// ---- DUTs/IO/Topology/Term_1047_EK1100_7ACEE53D.TcDUT
{attribute 'GeneratedUsingTerminal: EK1100-0000-0018'}
{attribute addProperty BoxType "EK1100-0000-0018"}
{attribute addProperty Id "Term_1048_EL1809EL1809_32157CFD20Term_1049_EL1809EL1809_32157CFD20Term_1050_EL1809EL1809_32157CFD20Term_1051_EL1809EL1809_32157CFD20Term_1052_EL1809EL1809_32157CFD20Term_1053_EL1809EL1809_32157CFD20Term_1054_EL1809EL1809_32157CFD20Term_1055_EL1809EL1809_32157CFD20Term_1056_EL1809EL1809_32157CFD20Term_1057_EL1809EL1809_32157CFD20Term_1058_EL1809EL1809_32157CFD20Term_1059_EL1809EL1809_32157CFD20Term_1060_EL1809EL1809_32157CFD20Term_1061_EL1809EL1809_32157CFD20Term_1062_EL1809EL1809_32157CFD20Term_1063_EL1809EL1809_32157CFD20Term_1064_EL1809EL1809_32157CFD20Term_1065_EL1809EL1809_32157CFD20Term_1066_EL1809EL1809_32157CFD20Term_1068_EL1809EL1809_32157CFD20Term_1069_EL1809EL1809_32157CFD20Term_1070_EL1809EL1809_32157CFD20Term_1072_EL1809EL1809_32157CFD20Term_1073_EL1809EL1809_32157CFD20Term_1076_EL1809EL1809_32157CFD20Term_1077_EL1809EL1809_32157CFD20Term_1078_EL1809EL1809_32157CFD20Term_1081_EL1809EL1809_32157CFD20Term_1082_EL1809EL1809_32157CFD20Term_1083_EL1809EL1809_32157CFD20Term_1084_EL1809EL1809_32157CFD20Term_1085_EL1809EL1809_32157CFD20Term_1086_EL1809EL1809_32157CFD20Term_1087_EL1809EL1809_32157CFD20Term_1088_EL1809EL1809_32157CFD20Term_1089_EL1809EL1809_32157CFD20Term_1090_EL1809EL1809_32157CFD20Term_1091_EL1809EL1809_32157CFD20Term_1092_EL1809EL1809_32157CFD20Term_1093_EL1809EL1809_32157CFD20Term_1094_EL1809EL1809_32157CFD20Term_1095_EL1809EL1809_32157CFD20Term_1096_EL1809EL1809_32157CFD20Term_1097_EL1809EL1809_32157CFD20Term_1098_EL1809EL1809_32157CFD20Term_1099_EL1809EL1809_32157CFD20Term_1100_EL1809EL1809_32157CFD20Term_1101_EL1809EL1809_32157CFD20Term_1102_EL1809EL1809_32157CFD20Term_1103_EL1809EL1809_32157CFD20Term_1104_EL1809EL1809_32157CFD20Term_1105_EL1809EL1809_32157CFD20Term_1106_EL1809EL1809_32157CFD20Term_1107_EL1809EL1809_32157CFD20Term_1108_EL1809EL1809_32157CFD20Term_1109_EL1809EL1809_32157CFD20Term_1110_EL1809EL1809_32157CFD20Term_1111_EL1809EL1809_32157CFD20Term_1112_EL1809EL1809_32157CFD20Term_1113_EL1809EL1809_32157CFD20Term_1114_EL1809EL1809_32157CFD20Term_1115_EL1809EL1809_32157CFD20Term_1116_EL1809EL1809_32157CFD20Term_1117_EL1809EL1809_32157CFD20Term_1118_EL1809EL1809_32157CFD20Term_1119_EL1809EL1809_32157CFD20Term_1120_EL1809EL1809_32157CFD20Term_1121_EL1809EL1809_32157CFD20Term_1122_EL1809EL1809_32157CFD20Term_1123_EL1809EL1809_32157CFD20Term_1124_EL1809EL1809_32157CFD20Term_1125_EL1809EL1809_32157CFD20Term_1126_EL1809EL1809_32157CFD20Term_1127_EL1809EL1809_32157CFD20Term_1128_EL1809EL1809_32157CFD20Term_1129_EL1809EL1809_32157CFD20Term_1130_EL1809EL1809_32157CFD20Term_1131_EL1809EL1809_32157CFD20Term_1132_EL1809EL1809_32157CFD20Term_1134_EL1809EL1809_32157CFD20Term_1135_EL1809EL1809_32157CFD20Term_1136_EL1809EL1809_32157CFD20Term_1137_EL1809EL1809_32157CFD20Term_1138_EL1809EL1809_32157CFD20Term_1139_EL1809EL1809_32157CFD20Term_1140_EL1809EL1809_32157CFD20Term_1141_EL1809EL1809_32157CFD20Term_1142_EL1809EL1809_32157CFD20Term_1143_EL1809EL1809_32157CFD20Term_1144_EL1809EL1809_32157CFD20Term_1145_EL1809EL1809_32157CFD20Term_1146_EL1809EL1809_32157CFD20Term_1147_EL1809EL1809_32157CFD20Term_1148_EL1809EL1809_32157CFD20Term_1149_EL1809EL1809_32157CFD20Term_1150_EL1809EL1809_32157CFD20Term_1151_EL1809EL1809_32157CFD20Term_1154_EL1809EL1809_32157CFD20Term_1155_EL1809EL1809_32157CFD20Term_1156_EL1809EL1809_32157CFD20Term_1157_EK1110EK1110_1FC0878B2"}
{attribute addProperty CRC "2060379453"}
{attribute addProperty Size "2002"}
{attribute addProperty Name "Term 1047 (EK1100)"}
TYPE Term_1047_EK1100_7ACEE53D EXTENDS EK1100_1FC0878B :
STRUCT
    {attribute addProperty Name "Term 1048 (EL1809)"}
    {attribute addProperty PreviousPort "Term 1047 (EK1100) : B"}
    {attribute addProperty SyncUnit "default"}
    Term_1048_EL1809 : EL1809_32157CFD;
    {attribute addProperty Name "Term 1049 (EL1809)"}
    {attribute addProperty PreviousPort "Term 1048 (EL1809) : B"}
    {attribute addProperty SyncUnit "default"}
    Term_1049_EL1809 : EL1809_32157CFD;
    {attribute addProperty Name "Term 1050 (EL1809)"}
    {attribute addProperty PreviousPort "Term 1049 (EL1809) : B"}
    {attribute addProperty SyncUnit "default"}
    Term_1050_EL1809 : EL1809_32157CFD;
    {attribute addProperty Name "Term 1051 (EL1809)"}
    {attribute addProperty PreviousPort "Term 1050 (EL1809) : B"}
    {attribute addProperty SyncUnit "default"}
    Term_1051_EL1809 : EL1809_32157CFD;
    {attribute addProperty Name "Term 1052 (EL1809)"}
    {attribute addProperty PreviousPort "Term 1051 (EL1809) : B"}
    {attribute addProperty SyncUnit "default"}
    Term_1052_EL1809 : EL1809_32157CFD;
    {attribute addProperty Name "Term 1053 (EL1809)"}
    {attribute addProperty PreviousPort "Term 1052 (EL1809) : B"}
    {attribute addProperty SyncUnit "default"}
    Term_1053_EL1809 : EL1809_32157CFD;
    {attribute addProperty Name "Term 1054 (EL1809)"}
    {attribute addProperty PreviousPort "Term 1053 (EL1809) : B"}
    {attribute addProperty SyncUnit "default"}
    Term_1054_EL1809 : EL1809_32157CFD;
    {attribute addProperty Name "Term 1055 (EL1809)"}
    {attribute addProperty PreviousPort "Term 1054 (EL1809) : B"}
    {attribute addProperty SyncUnit "default"}
    Term_1055_EL1809 : EL1809_32157CFD;
    {attribute addProperty Name "Term 1056 (EL1809)"}
    {attribute addProperty PreviousPort "Term 1055 (EL1809) : B"}
    {attribute addProperty SyncUnit "default"}
    Term_1056_EL1809 : EL1809_32157CFD;
    {attribute addProperty Name "Term 1057 (EL1809)"}
    {attribute addProperty PreviousPort "Term 1056 (EL1809) : B"}
    {attribute addProperty SyncUnit "default"}
    Term_1057_EL1809 : EL1809_32157CFD;
    {attribute addProperty Name "Term 1058 (EL1809)"}
    {attribute addProperty PreviousPort "Term 1057 (EL1809) : B"}
    {attribute addProperty SyncUnit "default"}
    Term_1058_EL1809 : EL1809_32157CFD;
    {attribute addProperty Name "Term 1059 (EL1809)"}
    {attribute addProperty PreviousPort "Term 1058 (EL1809) : B"}
    {attribute addProperty SyncUnit "default"}
    Term_1059_EL1809 : EL1809_32157CFD;
    {attribute addProperty Name "Term 1060 (EL1809)"}
    {attribute addProperty PreviousPort "Term 1059 (EL1809) : B"}
    {attribute addProperty SyncUnit "default"}
    Term_1060_EL1809 : EL1809_32157CFD;
    {attribute addProperty Name "Term 1061 (EL1809)"}
    {attribute addProperty PreviousPort "Term 1060 (EL1809) : B"}
    {attribute addProperty SyncUnit "default"}
    Term_1061_EL1809 : EL1809_32157CFD;
    {attribute addProperty Name "Term 1062 (EL1809)"}
    {attribute addProperty PreviousPort "Term 1061 (EL1809) : B"}
    {attribute addProperty SyncUnit "default"}
    Term_1062_EL1809 : EL1809_32157CFD;
    {attribute addProperty Name "Term 1063 (EL1809)"}
    {attribute addProperty PreviousPort "Term 1062 (EL1809) : B"}
    {attribute addProperty SyncUnit "default"}
    Term_1063_EL1809 : EL1809_32157CFD;
    {attribute addProperty Name "Term 1064 (EL1809)"}
    {attribute addProperty PreviousPort "Term 1063 (EL1809) : B"}
    {attribute addProperty SyncUnit "default"}
    Term_1064_EL1809 : EL1809_32157CFD;
    {attribute addProperty Name "Term 1065 (EL1809)"}
    {attribute addProperty PreviousPort "Term 1064 (EL1809) : B"}
    {attribute addProperty SyncUnit "default"}
    Term_1065_EL1809 : EL1809_32157CFD;
    {attribute addProperty Name "Term 1066 (EL1809)"}
    {attribute addProperty PreviousPort "Term 1065 (EL1809) : B"}
    {attribute addProperty SyncUnit "default"}
    Term_1066_EL1809 : EL1809_32157CFD;
    {attribute addProperty Name "Term 1068 (EL1809)"}
    {attribute addProperty PreviousPort "Term 1066 (EL1809) : B"}
    {attribute addProperty SyncUnit "default"}
    Term_1068_EL1809 : EL1809_32157CFD;
    {attribute addProperty Name "Term 1069 (EL1809)"}
    {attribute addProperty PreviousPort "Term 1068 (EL1809) : B"}
    {attribute addProperty SyncUnit "default"}
    Term_1069_EL1809 : EL1809_32157CFD;
    {attribute addProperty Name "Term 1070 (EL1809)"}
    {attribute addProperty PreviousPort "Term 1069 (EL1809) : B"}
    {attribute addProperty SyncUnit "default"}
    Term_1070_EL1809 : EL1809_32157CFD;
    {attribute addProperty Name "Term 1072 (EL1809)"}
    {attribute addProperty PreviousPort "Term 1070 (EL1809) : B"}
    {attribute addProperty SyncUnit "default"}
    Term_1072_EL1809 : EL1809_32157CFD;
    {attribute addProperty Name "Term 1073 (EL1809)"}
    {attribute addProperty PreviousPort "Term 1072 (EL1809) : B"}
    {attribute addProperty SyncUnit "default"}
    Term_1073_EL1809 : EL1809_32157CFD;
    {attribute addProperty Name "Term 1076 (EL1809)"}
    {attribute addProperty PreviousPort "Term 1073 (EL1809) : B"}
    {attribute addProperty SyncUnit "default"}
    Term_1076_EL1809 : EL1809_32157CFD;
    {attribute addProperty Name "Term 1077 (EL1809)"}
    {attribute addProperty PreviousPort "Term 1076 (EL1809) : B"}
    {attribute addProperty SyncUnit "default"}
    Term_1077_EL1809 : EL1809_32157CFD;
    {attribute addProperty Name "Term 1078 (EL1809)"}
    {attribute addProperty PreviousPort "Term 1077 (EL1809) : B"}
    {attribute addProperty SyncUnit "default"}
    Term_1078_EL1809 : EL1809_32157CFD;
    {attribute addProperty Name "Term 1081 (EL1809)"}
    {attribute addProperty PreviousPort "Term 1078 (EL1809) : B"}
    {attribute addProperty SyncUnit "default"}
    Term_1081_EL1809 : EL1809_32157CFD;
    {attribute addProperty Name "Term 1082 (EL1809)"}
    {attribute addProperty PreviousPort "Term 1081 (EL1809) : B"}
    {attribute addProperty SyncUnit "default"}
    Term_1082_EL1809 : EL1809_32157CFD;
    {attribute addProperty Name "Term 1083 (EL1809)"}
    {attribute addProperty PreviousPort "Term 1082 (EL1809) : B"}
    {attribute addProperty SyncUnit "default"}
    Term_1083_EL1809 : EL1809_32157CFD;
    {attribute addProperty Name "Term 1084 (EL1809)"}
    {attribute addProperty PreviousPort "Term 1083 (EL1809) : B"}
    {attribute addProperty SyncUnit "default"}
    Term_1084_EL1809 : EL1809_32157CFD;
    {attribute addProperty Name "Term 1085 (EL1809)"}
    {attribute addProperty PreviousPort "Term 1084 (EL1809) : B"}
    {attribute addProperty SyncUnit "default"}
    Term_1085_EL1809 : EL1809_32157CFD;
    {attribute addProperty Name "Term 1086 (EL1809)"}
    {attribute addProperty PreviousPort "Term 1085 (EL1809) : B"}
    {attribute addProperty SyncUnit "default"}
    Term_1086_EL1809 : EL1809_32157CFD;
    {attribute addProperty Name "Term 1087 (EL1809)"}
    {attribute addProperty PreviousPort "Term 1086 (EL1809) : B"}
    {attribute addProperty SyncUnit "default"}
    Term_1087_EL1809 : EL1809_32157CFD;
    {attribute addProperty Name "Term 1088 (EL1809)"}
    {attribute addProperty PreviousPort "Term 1087 (EL1809) : B"}
    {attribute addProperty SyncUnit "default"}
    Term_1088_EL1809 : EL1809_32157CFD;
    {attribute addProperty Name "Term 1089 (EL1809)"}
    {attribute addProperty PreviousPort "Term 1088 (EL1809) : B"}
    {attribute addProperty SyncUnit "default"}
    Term_1089_EL1809 : EL1809_32157CFD;
    {attribute addProperty Name "Term 1090 (EL1809)"}
    {attribute addProperty PreviousPort "Term 1089 (EL1809) : B"}
    {attribute addProperty SyncUnit "default"}
    Term_1090_EL1809 : EL1809_32157CFD;
    {attribute addProperty Name "Term 1091 (EL1809)"}
    {attribute addProperty PreviousPort "Term 1090 (EL1809) : B"}
    {attribute addProperty SyncUnit "default"}
    Term_1091_EL1809 : EL1809_32157CFD;
    {attribute addProperty Name "Term 1092 (EL1809)"}
    {attribute addProperty PreviousPort "Term 1091 (EL1809) : B"}
    {attribute addProperty SyncUnit "default"}
    Term_1092_EL1809 : EL1809_32157CFD;
    {attribute addProperty Name "Term 1093 (EL1809)"}
    {attribute addProperty PreviousPort "Term 1092 (EL1809) : B"}
    {attribute addProperty SyncUnit "default"}
    Term_1093_EL1809 : EL1809_32157CFD;
    {attribute addProperty Name "Term 1094 (EL1809)"}
    {attribute addProperty PreviousPort "Term 1093 (EL1809) : B"}
    {attribute addProperty SyncUnit "default"}
    Term_1094_EL1809 : EL1809_32157CFD;
    {attribute addProperty Name "Term 1095 (EL1809)"}
    {attribute addProperty PreviousPort "Term 1094 (EL1809) : B"}
    {attribute addProperty SyncUnit "default"}
    Term_1095_EL1809 : EL1809_32157CFD;
    {attribute addProperty Name "Term 1096 (EL1809)"}
    {attribute addProperty PreviousPort "Term 1095 (EL1809) : B"}
    {attribute addProperty SyncUnit "default"}
    Term_1096_EL1809 : EL1809_32157CFD;
    {attribute addProperty Name "Term 1097 (EL1809)"}
    {attribute addProperty PreviousPort "Term 1096 (EL1809) : B"}
    {attribute addProperty SyncUnit "default"}
    Term_1097_EL1809 : EL1809_32157CFD;
    {attribute addProperty Name "Term 1098 (EL1809)"}
    {attribute addProperty PreviousPort "Term 1097 (EL1809) : B"}
    {attribute addProperty SyncUnit "default"}
    Term_1098_EL1809 : EL1809_32157CFD;
    {attribute addProperty Name "Term 1099 (EL1809)"}
    {attribute addProperty PreviousPort "Term 1098 (EL1809) : B"}
    {attribute addProperty SyncUnit "default"}
    Term_1099_EL1809 : EL1809_32157CFD;
    {attribute addProperty Name "Term 1100 (EL1809)"}
    {attribute addProperty PreviousPort "Term 1099 (EL1809) : B"}
    {attribute addProperty SyncUnit "default"}
    Term_1100_EL1809 : EL1809_32157CFD;
    {attribute addProperty Name "Term 1101 (EL1809)"}
    {attribute addProperty PreviousPort "Term 1100 (EL1809) : B"}
    {attribute addProperty SyncUnit "default"}
    Term_1101_EL1809 : EL1809_32157CFD;
    {attribute addProperty Name "Term 1102 (EL1809)"}
    {attribute addProperty PreviousPort "Term 1101 (EL1809) : B"}
    {attribute addProperty SyncUnit "default"}
    Term_1102_EL1809 : EL1809_32157CFD;
    {attribute addProperty Name "Term 1103 (EL1809)"}
    {attribute addProperty PreviousPort "Term 1102 (EL1809) : B"}
    {attribute addProperty SyncUnit "default"}
    Term_1103_EL1809 : EL1809_32157CFD;
    {attribute addProperty Name "Term 1104 (EL1809)"}
    {attribute addProperty PreviousPort "Term 1103 (EL1809) : B"}
    {attribute addProperty SyncUnit "default"}
    Term_1104_EL1809 : EL1809_32157CFD;
    {attribute addProperty Name "Term 1105 (EL1809)"}
    {attribute addProperty PreviousPort "Term 1104 (EL1809) : B"}
    {attribute addProperty SyncUnit "default"}
    Term_1105_EL1809 : EL1809_32157CFD;
    {attribute addProperty Name "Term 1106 (EL1809)"}
    {attribute addProperty PreviousPort "Term 1105 (EL1809) : B"}
    {attribute addProperty SyncUnit "default"}
    Term_1106_EL1809 : EL1809_32157CFD;
    {attribute addProperty Name "Term 1107 (EL1809)"}
    {attribute addProperty PreviousPort "Term 1106 (EL1809) : B"}
    {attribute addProperty SyncUnit "default"}
    Term_1107_EL1809 : EL1809_32157CFD;
    {attribute addProperty Name "Term 1108 (EL1809)"}
    {attribute addProperty PreviousPort "Term 1107 (EL1809) : B"}
    {attribute addProperty SyncUnit "default"}
    Term_1108_EL1809 : EL1809_32157CFD;
    {attribute addProperty Name "Term 1109 (EL1809)"}
    {attribute addProperty PreviousPort "Term 1108 (EL1809) : B"}
    {attribute addProperty SyncUnit "default"}
    Term_1109_EL1809 : EL1809_32157CFD;
    {attribute addProperty Name "Term 1110 (EL1809)"}
    {attribute addProperty PreviousPort "Term 1109 (EL1809) : B"}
    {attribute addProperty SyncUnit "default"}
    Term_1110_EL1809 : EL1809_32157CFD;
    {attribute addProperty Name "Term 1111 (EL1809)"}
    {attribute addProperty PreviousPort "Term 1110 (EL1809) : B"}
    {attribute addProperty SyncUnit "default"}
    Term_1111_EL1809 : EL1809_32157CFD;
    {attribute addProperty Name "Term 1112 (EL1809)"}
    {attribute addProperty PreviousPort "Term 1111 (EL1809) : B"}
    {attribute addProperty SyncUnit "default"}
    Term_1112_EL1809 : EL1809_32157CFD;
    {attribute addProperty Name "Term 1113 (EL1809)"}
    {attribute addProperty PreviousPort "Term 1112 (EL1809) : B"}
    {attribute addProperty SyncUnit "default"}
    Term_1113_EL1809 : EL1809_32157CFD;
    {attribute addProperty Name "Term 1114 (EL1809)"}
    {attribute addProperty PreviousPort "Term 1113 (EL1809) : B"}
    {attribute addProperty SyncUnit "default"}
    Term_1114_EL1809 : EL1809_32157CFD;
    {attribute addProperty Name "Term 1115 (EL1809)"}
    {attribute addProperty PreviousPort "Term 1114 (EL1809) : B"}
    {attribute addProperty SyncUnit "default"}
    Term_1115_EL1809 : EL1809_32157CFD;
    {attribute addProperty Name "Term 1116 (EL1809)"}
    {attribute addProperty PreviousPort "Term 1115 (EL1809) : B"}
    {attribute addProperty SyncUnit "default"}
    Term_1116_EL1809 : EL1809_32157CFD;
    {attribute addProperty Name "Term 1117 (EL1809)"}
    {attribute addProperty PreviousPort "Term 1116 (EL1809) : B"}
    {attribute addProperty SyncUnit "default"}
    Term_1117_EL1809 : EL1809_32157CFD;
    {attribute addProperty Name "Term 1118 (EL1809)"}
    {attribute addProperty PreviousPort "Term 1117 (EL1809) : B"}
    {attribute addProperty SyncUnit "default"}
    Term_1118_EL1809 : EL1809_32157CFD;
    {attribute addProperty Name "Term 1119 (EL1809)"}
    {attribute addProperty PreviousPort "Term 1118 (EL1809) : B"}
    {attribute addProperty SyncUnit "default"}
    Term_1119_EL1809 : EL1809_32157CFD;
    {attribute addProperty Name "Term 1120 (EL1809)"}
    {attribute addProperty PreviousPort "Term 1119 (EL1809) : B"}
    {attribute addProperty SyncUnit "default"}
    Term_1120_EL1809 : EL1809_32157CFD;
    {attribute addProperty Name "Term 1121 (EL1809)"}
    {attribute addProperty PreviousPort "Term 1120 (EL1809) : B"}
    {attribute addProperty SyncUnit "default"}
    Term_1121_EL1809 : EL1809_32157CFD;
    {attribute addProperty Name "Term 1122 (EL1809)"}
    {attribute addProperty PreviousPort "Term 1121 (EL1809) : B"}
    {attribute addProperty SyncUnit "default"}
    Term_1122_EL1809 : EL1809_32157CFD;
    {attribute addProperty Name "Term 1123 (EL1809)"}
    {attribute addProperty PreviousPort "Term 1122 (EL1809) : B"}
    {attribute addProperty SyncUnit "default"}
    Term_1123_EL1809 : EL1809_32157CFD;
    {attribute addProperty Name "Term 1124 (EL1809)"}
    {attribute addProperty PreviousPort "Term 1123 (EL1809) : B"}
    {attribute addProperty SyncUnit "default"}
    Term_1124_EL1809 : EL1809_32157CFD;
    {attribute addProperty Name "Term 1125 (EL1809)"}
    {attribute addProperty PreviousPort "Term 1124 (EL1809) : B"}
    {attribute addProperty SyncUnit "default"}
    Term_1125_EL1809 : EL1809_32157CFD;
    {attribute addProperty Name "Term 1126 (EL1809)"}
    {attribute addProperty PreviousPort "Term 1125 (EL1809) : B"}
    {attribute addProperty SyncUnit "default"}
    Term_1126_EL1809 : EL1809_32157CFD;
    {attribute addProperty Name "Term 1127 (EL1809)"}
    {attribute addProperty PreviousPort "Term 1126 (EL1809) : B"}
    {attribute addProperty SyncUnit "default"}
    Term_1127_EL1809 : EL1809_32157CFD;
    {attribute addProperty Name "Term 1128 (EL1809)"}
    {attribute addProperty PreviousPort "Term 1127 (EL1809) : B"}
    {attribute addProperty SyncUnit "default"}
    Term_1128_EL1809 : EL1809_32157CFD;
    {attribute addProperty Name "Term 1129 (EL1809)"}
    {attribute addProperty PreviousPort "Term 1128 (EL1809) : B"}
    {attribute addProperty SyncUnit "default"}
    Term_1129_EL1809 : EL1809_32157CFD;
    {attribute addProperty Name "Term 1130 (EL1809)"}
    {attribute addProperty PreviousPort "Term 1129 (EL1809) : B"}
    {attribute addProperty SyncUnit "default"}
    Term_1130_EL1809 : EL1809_32157CFD;
    {attribute addProperty Name "Term 1131 (EL1809)"}
    {attribute addProperty PreviousPort "Term 1130 (EL1809) : B"}
    {attribute addProperty SyncUnit "default"}
    Term_1131_EL1809 : EL1809_32157CFD;
    {attribute addProperty Name "Term 1132 (EL1809)"}
    {attribute addProperty PreviousPort "Term 1131 (EL1809) : B"}
    {attribute addProperty SyncUnit "default"}
    Term_1132_EL1809 : EL1809_32157CFD;
    {attribute addProperty Name "Term 1134 (EL1809)"}
    {attribute addProperty PreviousPort "Term 1132 (EL1809) : B"}
    {attribute addProperty SyncUnit "default"}
    Term_1134_EL1809 : EL1809_32157CFD;
    {attribute addProperty Name "Term 1135 (EL1809)"}
    {attribute addProperty PreviousPort "Term 1134 (EL1809) : B"}
    {attribute addProperty SyncUnit "default"}
    Term_1135_EL1809 : EL1809_32157CFD;
    {attribute addProperty Name "Term 1136 (EL1809)"}
    {attribute addProperty PreviousPort "Term 1135 (EL1809) : B"}
    {attribute addProperty SyncUnit "default"}
    Term_1136_EL1809 : EL1809_32157CFD;
    {attribute addProperty Name "Term 1137 (EL1809)"}
    {attribute addProperty PreviousPort "Term 1136 (EL1809) : B"}
    {attribute addProperty SyncUnit "default"}
    Term_1137_EL1809 : EL1809_32157CFD;
    {attribute addProperty Name "Term 1138 (EL1809)"}
    {attribute addProperty PreviousPort "Term 1137 (EL1809) : B"}
    {attribute addProperty SyncUnit "default"}
    Term_1138_EL1809 : EL1809_32157CFD;
    {attribute addProperty Name "Term 1139 (EL1809)"}
    {attribute addProperty PreviousPort "Term 1138 (EL1809) : B"}
    {attribute addProperty SyncUnit "default"}
    Term_1139_EL1809 : EL1809_32157CFD;
    {attribute addProperty Name "Term 1140 (EL1809)"}
    {attribute addProperty PreviousPort "Term 1139 (EL1809) : B"}
    {attribute addProperty SyncUnit "default"}
    Term_1140_EL1809 : EL1809_32157CFD;
    {attribute addProperty Name "Term 1141 (EL1809)"}
    {attribute addProperty PreviousPort "Term 1140 (EL1809) : B"}
    {attribute addProperty SyncUnit "default"}
    Term_1141_EL1809 : EL1809_32157CFD;
    {attribute addProperty Name "Term 1142 (EL1809)"}
    {attribute addProperty PreviousPort "Term 1141 (EL1809) : B"}
    {attribute addProperty SyncUnit "default"}
    Term_1142_EL1809 : EL1809_32157CFD;
    {attribute addProperty Name "Term 1143 (EL1809)"}
    {attribute addProperty PreviousPort "Term 1142 (EL1809) : B"}
    {attribute addProperty SyncUnit "default"}
    Term_1143_EL1809 : EL1809_32157CFD;
    {attribute addProperty Name "Term 1144 (EL1809)"}
    {attribute addProperty PreviousPort "Term 1143 (EL1809) : B"}
    {attribute addProperty SyncUnit "default"}
    Term_1144_EL1809 : EL1809_32157CFD;
    {attribute addProperty Name "Term 1145 (EL1809)"}
    {attribute addProperty PreviousPort "Term 1144 (EL1809) : B"}
    {attribute addProperty SyncUnit "default"}
    Term_1145_EL1809 : EL1809_32157CFD;
    {attribute addProperty Name "Term 1146 (EL1809)"}
    {attribute addProperty PreviousPort "Term 1145 (EL1809) : B"}
    {attribute addProperty SyncUnit "default"}
    Term_1146_EL1809 : EL1809_32157CFD;
    {attribute addProperty Name "Term 1147 (EL1809)"}
    {attribute addProperty PreviousPort "Term 1146 (EL1809) : B"}
    {attribute addProperty SyncUnit "default"}
    Term_1147_EL1809 : EL1809_32157CFD;
    {attribute addProperty Name "Term 1148 (EL1809)"}
    {attribute addProperty PreviousPort "Term 1147 (EL1809) : B"}
    {attribute addProperty SyncUnit "default"}
    Term_1148_EL1809 : EL1809_32157CFD;
    {attribute addProperty Name "Term 1149 (EL1809)"}
    {attribute addProperty PreviousPort "Term 1148 (EL1809) : B"}
    {attribute addProperty SyncUnit "default"}
    Term_1149_EL1809 : EL1809_32157CFD;
    {attribute addProperty Name "Term 1150 (EL1809)"}
    {attribute addProperty PreviousPort "Term 1149 (EL1809) : B"}
    {attribute addProperty SyncUnit "default"}
    Term_1150_EL1809 : EL1809_32157CFD;
    {attribute addProperty Name "Term 1151 (EL1809)"}
    {attribute addProperty PreviousPort "Term 1150 (EL1809) : B"}
    {attribute addProperty SyncUnit "default"}
    Term_1151_EL1809 : EL1809_32157CFD;
    {attribute addProperty Name "Term 1154 (EL1809)"}
    {attribute addProperty PreviousPort "Term 1151 (EL1809) : B"}
    {attribute addProperty SyncUnit "default"}
    Term_1154_EL1809 : EL1809_32157CFD;
    {attribute addProperty Name "Term 1155 (EL1809)"}
    {attribute addProperty PreviousPort "Term 1154 (EL1809) : B"}
    {attribute addProperty SyncUnit "default"}
    Term_1155_EL1809 : EL1809_32157CFD;
    {attribute addProperty Name "Term 1156 (EL1809)"}
    {attribute addProperty PreviousPort "Term 1155 (EL1809) : B"}
    {attribute addProperty SyncUnit "default"}
    Term_1156_EL1809 : EL1809_32157CFD;
    {attribute addProperty Name "Term 1157 (EK1110)"}
    {attribute addProperty PreviousPort "Term 1156 (EL1809) : B"}
    {attribute addProperty SyncUnit "default"}
    Term_1157_EK1110 : EK1110_1FC0878B;
END_STRUCT
END_TYPE

// ---- DUTs/IO/Topology/Device_5_EtherCAT_0A694E3C.TcDUT
{attribute 'GeneratedUsingTerminal: IODEVICETYPE_ETHERCATPROT'}
{attribute addProperty BoxType "IODEVICETYPE_ETHERCATPROT"}
{attribute addProperty Id "Term_279_EK1100Term_279_EK1100_ED7D62722002Term_554_EK1100Term_554_EK1100_B580E2182002Term_748_EK1100Term_748_EK1100_BC4343B12002Term_881_EK1100Term_881_EK1100_F732F3702002Term_1047_EK1100Term_1047_EK1100_7ACEE53D2002SyncUnitsSyncUnits_C3A34B5018InputsInputs_A65FACA410OutputsOutputs_23C0ED1D6InfoDataInfoData_84133AC922"}
{attribute addProperty CRC "174673468"}
{attribute addProperty Size "10066"}
{attribute addProperty Name "Device 5 (EtherCAT)"}
TYPE Device_5_EtherCAT_0A694E3C EXTENDS TcoIo.EtcMasterBase_62654B43 :
STRUCT
    {attribute addProperty Name "Term 279 (EK1100)"}
    {attribute addProperty PreviousPort "Device 5 (EtherCAT) : Master"}
    {attribute addProperty SyncUnit "default"}
    Term_279_EK1100 : Term_279_EK1100_ED7D6272;
    {attribute addProperty Name "Term 554 (EK1100)"}
    {attribute addProperty PreviousPort "Term 495 (EK1110) : B"}
    {attribute addProperty SyncUnit "default"}
    Term_554_EK1100 : Term_554_EK1100_B580E218;
    {attribute addProperty Name "Term 748 (EK1100)"}
    {attribute addProperty PreviousPort "Term 747 (EK1110) : B"}
    {attribute addProperty SyncUnit "default"}
    Term_748_EK1100 : Term_748_EK1100_BC4343B1;
    {attribute addProperty Name "Term 881 (EK1100)"}
    {attribute addProperty PreviousPort "Term 880 (EK1110) : B"}
    {attribute addProperty SyncUnit "default"}
    Term_881_EK1100 : Term_881_EK1100_F732F370;
    {attribute addProperty Name "Term 1047 (EK1100)"}
    {attribute addProperty PreviousPort "Term 1046 (EK1110) : B"}
    {attribute addProperty SyncUnit "default"}
    Term_1047_EK1100 : Term_1047_EK1100_7ACEE53D;
    {attribute addProperty Name "SyncUnits"}
    SyncUnits : SyncUnits_C3A34B50;
    {attribute addProperty Name "Inputs"}
    Inputs : TcoIo.Inputs_A65FACA4;
    {attribute addProperty Name "Outputs"}
    Outputs : TcoIo.Outputs_23C0ED1D;
    {attribute addProperty Name "InfoData"}
    InfoData : TcoIo.InfoData_84133AC9;
END_STRUCT
END_TYPE

// ---- GVLs/GVL_iXlinker.TcGVL
{attribute 'qualified_only'}
VAR_GLOBAL
    Device_1_EtherCAT : Device_1_EtherCAT_49C09C66;
    Device_2_EtherCAT : Device_2_EtherCAT_22CD061B;
    Device_3_EtherCAT : Device_3_EtherCAT_368E547E;
    //		Device_4_EtherCAT : Device_4_EtherCAT_07442C6B;
    //		Device_5_EtherCAT : Device_5_EtherCAT_0A694E3C;
END_VAR

// ---- POUs/MAIN.TcPOU
PROGRAM MAIN
VAR
    _tcc : tcc;
END_VAR

_tcc.Run();

END_PROGRAM

// ---- POUs/tcc.TcPOU
FUNCTION_BLOCK tcc EXTENDS TcoCore.TcoContext
VAR
    {attribute addProperty Name "Device 1 (EtherCAT)"}
    Device_1 : TcoIo.TcoEthercatMasterDevice(THIS^);
    {attribute addProperty Name "Device 2 (EtherCAT)"}
    Device_2 : TcoIo.TcoEthercatMasterDevice(THIS^);
    {attribute addProperty Name "EtherCAT component"}
    EcatComponent : TestEcatComponent(THIS^);
END_VAR

{attribute 'hide'}
METHOD FB_init : BOOL
VAR_INPUT
    bInitRetains : BOOL; // if TRUE, the retain variables are initialized (warm start / cold start)
    bInCopyCode : BOOL; // if TRUE, the instance afterwards gets moved into the copy code (online change)
END_VAR
END_METHOD

(*~
    <docu>
        <summary>
            Main method of the TcoContext. This is the entry point of any control logic that belongs to this context.
            The call of this method is ensured by calling the <c>InstanceName.Run()</c> method, and it must not be called explicitly.
            This method is abstract, and it must be overridden in derived block.
        </summary>
    </docu>
~*)
METHOD PROTECTED Main
VAR
    ams : AMSADDR;
END_VAR
Device_1(SyncUnits := ADR(GVL_iXlinker.Device_1_EtherCAT.SyncUnits),
    SyncUnitsSize := SIZEOF(GVL_iXlinker.Device_1_EtherCAT.SyncUnits),
    Inputs := GVL_iXlinker.Device_1_EtherCAT.Inputs,
    InfoData := GVL_iXlinker.Device_1_EtherCAT.InfoData);

Device_2(SyncUnits := ADR(GVL_iXlinker.Device_2_EtherCAT.SyncUnits),
    SyncUnitsSize := SIZEOF(GVL_iXlinker.Device_2_EtherCAT.SyncUnits),
    Inputs := GVL_iXlinker.Device_2_EtherCAT.Inputs,
    InfoData := GVL_iXlinker.Device_2_EtherCAT.InfoData);

EcatComponent(AdsAddr := ams);
EcatComponent.Service();
END_METHOD

END_FUNCTION_BLOCK

// ---- POUs/TestEcatComponent.TcPOU
FUNCTION_BLOCK PUBLIC TestEcatComponent EXTENDS TcoIo.TcoEcatComponent
VAR_OUTPUT
END_VAR
VAR
END_VAR

SUPER^(AdsAddr := AdsAddr);

END_FUNCTION_BLOCK
